PROGRAM MAIN
VAR
	motor1 : MotorPositionController;
	motor_param : MotorPositionController.MotorParam;
	motor_data : MotorPositionController.MotorData;
	motor_state : MotorPositionController.MotorState;
	
	sensor_data : SensorData;
END_VAR

motor1(motor_axis:= GVL.axis1, motor_param:= motor_param, motor_data=> motor_data, motor_state=> motor_state);

END_PROGRAM

(* stored: Version 1.1.0.1, ProductVersion 3.1.4024.11
   POU MAIN: Id {13aa0b6a-1832-4149-b405-c6ea458a212e}, SpecialFunc None *)
